(*======================================================================================================================================*)
(*//=============================================================================\\
||  _   _ _  __  _         _                        _   _                      ||
|| | \ | | |/ / / \  _   _| |_ ___  _ __ ___   __ _| |_(_) ___  _ __         ||
|| |  \| | ' / / _ \| | | | __/ _ \| '_ ` _ \ / _` | __| |/ _ \| '_ \        ||
|| | |\  | . \/ ___ \ |_| | || (_) | | | | | | (_| | |_| | (_) | | | |       ||
|| |_| \_|_|\_\_/  \_\__,_|\__\___/|_| |_| |_|\__,_|\__|_|\___/|_| |_|       ||
||                                                                             ||
\\=============================================================================//
fb_BusDimmEvent:	Dieser Baustein sieht Dimmer Events und wertet diese aus, möglichst effizient.
								  *)
(*
Date          	| Version    	| created under        	| Author          	| Remark *)
(*====================================================================================================================================================*)
(*13/01/2026   	| 1.00      		| TC3		  		| N.Kersting       | first release *)
(*25/01/2026   	| 2.00      		| TC3		  		| N.Kersting       | Suchstring umstellung auf ASCII_RS485 Funktion *)
(*====================================================================================================================================================*)
FUNCTION_BLOCK fb_BusDimmEvent
VAR_INPUT
	 I_bExecute				:BOOL := TRUE;	// Aktiviert den Baustein 
	 I_bReset				:BOOL;
	 I_diID        			:DINT;     // Geräte-ID (z.B. '12345')
	 I_iInstID				:INT 	:=	17;
	 I_sReceivedString		:STRING(255);	
END_VAR
VAR_OUTPUT
	Q_iOut					:ARRAY[1..6] OF  INT;
	Q_bStartupDone			:BOOL;
END_VAR
VAR
	i						:INT;
	findString0				:ARRAY[1..6] OF STRING(255);
	
	iFindString				:ARRAY[1..6] OF INT;
	startPos 				:ARRAY[1..6] OF INT;
	
	bStartupStart			:BOOL;
	bStartupDone			:BOOL;
	
	iStartup				:INT;
	
	sLastString				:STRING(255);
	bNeedProcess			:BOOL;
END_VAR

(* Automatische Fehlererkennung *)
IF NOT I_bExecute
	OR (I_diID = 0)
	OR (I_iInstID = 0)
THEN
	iStartup := 0;
END_IF

(* Warten, ob der String sich geändert hat*)
bNeedProcess :=	(I_sReceivedString <> sLastString) 
				AND (I_sReceivedString <> '');

CASE iStartup OF 
(*=====================================*)
0 :	(* INIT *)
	bStartupDone := FALSE;
	bStartupStart := FALSE;
	bNeedProcess := FALSE;
	sLastString := '';
	
	FOR i := 1 TO 6 BY 1 DO
		
		Q_iOut[i] := 0;
		
	END_FOR	
	
	IF I_bExecute
		AND NOT bStartupDone
		AND NOT I_bReset
		AND (I_diID <> 0)
		AND (I_iInstID <>0)
	THEN
		i := 1;
		bStartupStart := TRUE;
		iStartup := iStartup +10;
	END_IF
	
(*=====================================*)
10 :(* String vorbereiten *)	
		
	FOR i := 1 TO 6 BY 1 DO
		findString0[i] := F_RS485HB_TO_ASCII_RX(
							I_diID			:= I_diID, 
							I_iInstID		:= I_iInstID+i-1,	
							I_EnumHBUnitTX	:= E_EnumHBUnitTX.E_HB_UNIT_DIM, 	
							I_EnumHBCmdRX	:= E_EnumHBCmdRX.E_HB_CMD_rSTATUS , 
							I_iP1			:= 0);
	END_FOR
	
	
	IF i >= 6 THEN
		bStartupStart := FALSE;
		iStartup := 999;
	END_IF
	
(*=====================================*)
999 :(* READY *)
	bStartupDone := TRUE;
	
	IF I_bReset 
	THEN
		iStartup := 0;
	ELSE
		IF bNeedProcess
		THEN
			FOR i := 1 TO 6 BY 1 DO					
				iFindString[i] :=	FIND(I_sReceivedString,findString0[i]);
			
				IF iFindString[i]>0
				THEN
					startPos[i] := iFindString[i]; // Position des Suchstrings       
					(*Dimmer steht direkt nach dem Suchstring*)
					startPos[i] := startPos[i] + LEN(findString0[i]); (*Startposition für Temperatur*)
					(* Dimmer bis zum nächsten Komma oder Ende auslesen (maximal 6 Zeichen: z.B. 100)*)
					Q_iOut[i] := STRING_TO_INT(MID(I_sReceivedString, 3, startPos[i]));
				END_IF
			END_FOR	
			sLastString :=	I_sReceivedString;	(* Letzten String Speichern *)
		END_IF
	END_IF
END_CASE

Q_bStartupDone := bStartupDone;

END_FUNCTION_BLOCK

(* stored: Version 1.1.0.1, ProductVersion 3.1.4024.16
   POU fb_BusDimmEvent: Id {0af3948f-e53b-42ef-a663-182ad8a04da5}, SpecialFunc None *)
